// Mitsubishi GX Works2 project: 機電整合乙級第五題-ST   PLC: FX3U/FX3UC

// task Task_01 (event TRUE, interval 0, priority 31): POU_01

PROGRAM POU_01
VAR
  wProgramStep : INT;
  ldStore : R_TRIG;
  ldFetch : R_TRIG;
  wHighSpeed : INT;
  wLowSpeed : INT;
  wXPos : INT;
  tdT22 : TON;
END_VAR
VAR CONSTANT
  dwLEVEL1 : INT := 100;
END_VAR
VAR
  tdT23 : TON;
  wCellNo : INT;
  rtX10 : R_TRIG;
  tdT27 : TON;
  wZPos : INT;
  tdT29 : TON;
  ftX10 : F_TRIG;
  tdT33 : TON;
  tdT41 : TON;
  tdT42 : TON;
  tdT43 : TON;
  bOutbound : BOOL;
  tdT21 : TON;
  wXNext : INT;
  wXCurr : INT;
  bM17 : BOOL;
  bM143 : BOOL;
  tdT143 : TON;
  tdT144 : TON;
END_VAR
(* 機電整合乙級術科第五題
   Author: Steven Luo
   Date: 2018/10/25
*)

IF M8000 THEN
	WR3A(TRUE, 0, 21, D53);
	M8026 := TRUE;
END_IF;

IF M8002 THEN
	OUT_C(TRUE, CC251, K999999);
	wLowSpeed := 1200;
	wHighSpeed := 4000;
	D53 := wLowSpeed;
	wProgramStep := 0;
END_IF;

IF NOT X17 THEN (* 急停 *)
	ZRST(TRUE, Y0, Y7);
	ZRST(TRUE, D0, D50);
	ZRST(TRUE, M130, M144);
	ZRST(TRUE, M150, M153);
	D5 := 513;
	bM17 := TRUE;
	wProgramStep := 0;
END_IF;

IF X17 AND bM17 AND M132 THEN (* 解除急停，按下復歸 *)
	bM17 := FALSE;
	bM143 := TRUE;
	tdT143(IN := FALSE);
	tdT144(IN := FALSE);
	wProgramStep := 100;
END_IF;

IF bM143 THEN (* 黃燈閃爍 *)
	tdT143(IN := NOT tdT144.Q, PT := T#500ms);
	tdT144(IN := tdT143.Q, PT := T#500ms);
	M143 := tdT143.Q;
END_IF;

CASE wProgramStep OF
0:
	IF X17 THEN
		IF M130 THEN
			wProgramStep := 200;
		ELSE
			wProgramStep := 20;
		END_IF;
	END_IF;
20:
	IF M130 THEN
		wProgramStep := 0;
	END_IF;
	IF WORD_TO_INT(D0) > 0 THEN
		ldStore(_CLK := M135);
		ldFetch(_CLK := M136);
		IF ldStore.Q THEN
			IF D10 = 0 THEN
				D10 := D0;
			ELSIF (D11 = 0) AND (D0 <> D10) THEN
				D11 := D0;
			ELSIF (D12 = 0) AND (D0 <> D10) AND (D0 <> D11) THEN
				D12 := D0;
			END_IF;
			D0 := 0;
		END_IF;
		IF ldFetch.Q THEN
			IF D30 = 0 THEN
				D30 := D0;
			ELSIF (D31 = 0) AND (D0 <> D30) THEN
				D31 := D0;
			ELSIF (D32 = 0) AND (D0 <> D30) AND (D0 <> D31) THEN
				D32 := D0;
			END_IF;
			D0 := 0;
		END_IF;
	END_IF;
	IF M137 THEN
		D10 := 0;
		D11 := 0;
		D12 := 0;
		M152 := FALSE;
	END_IF;
	IF M138 THEN
		D30 := 0;
		D31 := 0;
		D32 := 0;
		M153 := FALSE;
	END_IF;
	IF M150 AND WORD_TO_INT(D10) > 0 THEN
		M152 := TRUE;
		M153 := FALSE;
	END_IF;
	IF M151 AND WORD_TO_INT(D30) > 0 THEN
		M152 := FALSE;
		M153 := TRUE;
	END_IF;
	IF X2 AND X4 AND X5 AND X6 THEN (* 原點條件 *)
		D5 := 0;
		IF M131 THEN
			wXPos := 0;
			wZPos := 0;
			wCellNo := 0;
			wXCurr := 0;
			tdT21(IN := FALSE);
			tdT22(IN := FALSE);
			tdT23(IN := FALSE);
			tdT27(IN := FALSE);
			tdT29(IN := FALSE);
			tdT33(IN := FALSE);
			tdT41(IN := FALSE);
			tdT42(IN := FALSE);
			tdT43(IN := FALSE);
			D5 := 510;
			IF M152 THEN (* 存料 *)
				wProgramStep := 21;
			ELSIF M153 THEN (* 取料 *)
				wProgramStep := 40;
			END_IF;
		END_IF;
	END_IF;
21:
	Y11 := TRUE;
	IF X3 THEN (* 進料感測 *)
		Y11 := FALSE;
		tdT21(IN := TRUE, PT := T#500ms);
		IF tdT21.Q THEN
			wProgramStep := 22;
		END_IF;
	END_IF;
22:
	Y6 := TRUE; (* Y軸伸前 *)
	IF X7 THEN (* Y軸前位 *)
		D5 := 511;
		Y7 := TRUE; (* D+氣壓夾爪夾 *)
		tdT22(IN := TRUE, PT := T#500ms);
		IF tdT22.Q THEN
			wProgramStep := 23;
		END_IF;
	END_IF;
23:
	Y3 := TRUE; (* Z軸上升 *)
	tdT23(IN := TRUE, PT := T#500ms);
	IF tdT23.Q THEN
		Y3 := FALSE;
		wProgramStep := 24;
	END_IF;
24:
	Y6 := FALSE; (* Y軸縮回 *)
	IF X6 THEN (* Y軸後位 *)
		D5 := 0;
		wProgramStep := 25;
	END_IF;
25:
	Y5 := TRUE; (* Z軸下降 *)
	IF X5 THEN
		Y5 := FALSE;
		wProgramStep := 26;
	END_IF;
26:
	IF WORD_TO_INT(D10) > 0 THEN
		wCellNo := D10;
		D10 := 0;
	ELSIF WORD_TO_INT(D11) > 0 THEN
		wCellNo := D11;
		D11 := 0;
	ELSIF WORD_TO_INT(D12) > 0 THEN
		wCellNo := D12;
		D12 := 0;
	END_IF;
	wXPos := wCellNo MOD 10;
	(* Z軸座標為C251數值 *)
	wZPos := dwLEVEL1 + (wCellNo / 10 - 1) * 1600;
	IF wXPos > 0 THEN
		D60 := 0;
		wProgramStep := 27;
	ELSE
		wProgramStep := 20;
	END_IF;
27:
	Y0 := TRUE; (* X軸右移 *)
	rtX10( _CLK := X10);
	IF rtX10.Q THEN
		wXPos := wXPos - 1;
	END_IF;
	IF wXPos = 1 THEN
		RAMP(TRUE, wHighSpeed, wLowSpeed, 50, D53);
	ELSIF wXPos = 0 THEN
		Y0 := FALSE;
		Y1 := TRUE; (* X軸停止 *)
		tdT27(IN := TRUE, PT := T#500ms);
		IF tdT27.Q THEN
			Y1 := FALSE;
			wProgramStep := 28;
		END_IF;
	ELSE
		RAMP(TRUE, wLowSpeed, wHighSpeed, 50, D60);
		D53 := D60;
	END_IF;
28:
	Y3 := TRUE; (* Z軸上升 *)
	IF CN251 >= INT_TO_DINT(wZPos) THEN
		Y3 := FALSE;
		IF M152 THEN
			wProgramStep := 29;
		ELSIF M153 THEN
			wProgramStep := 41;
		END_IF;
	END_IF;
29:
	Y6 := TRUE; (* Y軸伸前 *)
	IF X7 THEN (* Y軸前位 *)
		D5 := 511;
		Y7 := FALSE;
		Y10 := TRUE; (* D-氣壓夾爪放 *)
		tdT29(IN := TRUE, PT := T#300ms);
		IF tdT29.Q THEN
			Y10 := FALSE;
			IF M153 THEN
				bOutbound := TRUE;
			END_IF;
			wProgramStep := 30;
		END_IF;
	END_IF;
30:
	Y6 := FALSE; (* Y軸縮回 *)
	IF X6 THEN (* Y軸後位 *)
		D5 := 0;
		D60 := 0;
		IF M152 THEN
			wProgramStep := 31;
		ELSIF M153 THEN
			IF bOutbound THEN
				wProgramStep := 44;
			ELSE
				wProgramStep := 31;
			END_IF;
		END_IF;
	END_IF;
31:
	Y5 := TRUE; (* Z軸下降 *)
	IF X5 THEN
		Y5 := FALSE;
		wXPos := wCellNo MOD 10;
		IF M152 THEN
			wProgramStep := 32;
		ELSIF M153 THEN
			wXPos := (5 - wXPos) + 1;
			wProgramStep := 42;
		END_IF;
	END_IF;
32:
	Y2 := TRUE; (* X軸左移 *)
	ftX10(_CLK := X10);
	IF ftX10.Q THEN
		wXPos := wXPos - 1;
	END_IF;
	IF wXPos = 0 THEN
		RAMP(TRUE, wHighSpeed, wLowSpeed, 50, D53);
	ELSE
		RAMP(TRUE, wLowSpeed, wHighSpeed, 50, D60);
		D53 := D60;
	END_IF;
	IF X4 THEN
		Y2 := FALSE;
		Y1 := TRUE; (* X軸停止 *)
		wProgramStep := 33;
	END_IF;
33:
	tdT33(IN := TRUE, PT := T#300ms);
	IF tdT33.Q THEN
		Y1 := FALSE;
		tdT21(IN := FALSE);
		tdT22(IN := FALSE);
		tdT23(IN := FALSE);
		tdT27(IN := FALSE);
		tdT29(IN := FALSE);
		tdT33(IN := FALSE);
		tdT41(IN := FALSE);
		tdT42(IN := FALSE);
		tdT43(IN := FALSE);
		IF M152 THEN
			IF (D10 = 0) AND (D11 = 0) AND (D12 = 0) THEN
				wProgramStep := 34;
			ELSE
				wProgramStep := 21; (* 繼續進料 *)
			END_IF;
		ELSIF M153 THEN
			IF (D30 = 0) AND (D31 = 0) AND (D32 = 0) THEN
				M153 := FALSE;
				wProgramStep := 20;
			ELSE
				wProgramStep := 40; (* 繼續出料 *)
			END_IF;
		END_IF;
	END_IF;
34:
	Y12 := TRUE; (* 進料座下降 *)
	IF X2 THEN (* 進料原點極限 *)
		Y12 := FALSE;
		M152 := FALSE;
		wProgramStep := 20;
	END_IF;
40:
	IF WORD_TO_INT(D30) > 0 THEN
		wCellNo := D30;
		IF WORD_TO_INT(D31) > 0 THEN
			wXNext := D31;
		ELSE
			wXNext := 0;
		END_IF;
		D30 := 0;
	ELSIF WORD_TO_INT(D31) > 0 THEN
		wCellNo := D31;
		IF WORD_TO_INT(D32) > 0 THEN
			wXNext := D32;
		ELSE
			wXNext := 0;
		END_IF;
		D31 := 0;
	ELSIF WORD_TO_INT(D32) > 0 THEN
		wCellNo := D32;
		wXNext := 0;
		D32 := 0;
	END_IF;
	wXPos := wCellNo MOD 10 - wXCurr;
	(* Z軸座標為C251數值 *)
	wZPos := dwLEVEL1 + (wCellNo / 10 - 1) * 1600 - 100;
	IF wCellNo > 0 THEN
		D60 := 0;
		bOutbound := FALSE;
		wProgramStep := 27;
	ELSE
		wProgramStep := 20;
	END_IF;
41:
	Y6 := TRUE; (* Y軸伸前 *)
	IF X7 THEN (* Y軸前位 *)
		D5 := 511;
		Y7 := TRUE; (* D+氣壓夾爪夾 *)
		tdT41(IN := TRUE, PT := T#300ms);
		IF tdT41.Q THEN
			wProgramStep := 30;
		END_IF;
	END_IF;
42:
	Y3 := TRUE; (* Z軸上升 *)
	tdT42(IN := TRUE, PT := T#1s);
	IF tdT42.Q THEN
		Y3 := FALSE;
		wProgramStep := 43;
	END_IF;
43:
	Y0 := TRUE; (* X軸右移 *)
	ftX10( _CLK := X10);
	IF ftX10.Q THEN
		wXPos := wXPos - 1;
	END_IF;
	IF wXPos = 1 THEN
		RAMP(TRUE, wHighSpeed, wLowSpeed, 50, D53);
	ELSIF wXPos = 0 THEN
		Y0 := FALSE;
		Y1 := TRUE; (* X軸停止 *)
		tdT43(IN := TRUE, PT := T#500ms);
		IF tdT43.Q THEN
			Y1 := FALSE;
			wProgramStep := 29;
		END_IF;
	ELSE
		RAMP(TRUE, wLowSpeed, wHighSpeed, 50, D60);
		D53 := D60;
	END_IF;
44:
	Y5 := TRUE; (* Z軸下降 *)
	IF X5 THEN
		Y5 := FALSE;
		wXCurr := wXNext MOD 10;
		wXPos := 6 - wXCurr;
		IF wXNext = 0 THEN
			wProgramStep := 32;
		ELSE
			wProgramStep := 45;
		END_IF;
	END_IF;
45:
	Y2 := TRUE; (* X軸左移 *)
	rtX10( _CLK := X10);
	IF rtX10.Q THEN
		wXPos := wXPos - 1;
	END_IF;
	IF wXPos = 1 THEN
		RAMP(TRUE, wHighSpeed, wLowSpeed, 50, D53);
	ELSIF wXPos = 0 THEN
		Y2 := FALSE;
		Y1 := TRUE; (* X軸停止 *)
		tdT43(IN := TRUE, PT := T#500ms);
		IF tdT43.Q THEN
			Y1 := FALSE;
			wProgramStep := 33;
		END_IF;
	ELSE
		RAMP(TRUE, wLowSpeed, wHighSpeed, 50, D60);
		D53 := D60;
	END_IF;
100:
	D5 := 512;
	D53 := wLowSpeed;
	Y6 := FALSE;
	IF X6 THEN
		Y5 := TRUE;
		IF X5 THEN
			Y5 := FALSE;
			Y2 := TRUE;
			IF X4 THEN
				Y2 := FALSE;
				Y12 := TRUE;
				IF X2 THEN
					Y12 := FALSE;
					D5 := 0;
					bM143 := FALSE;
					M143 := FALSE;
					wProgramStep := 0;
				END_IF;
			END_IF;
		END_IF;
	END_IF;
200:
	IF X6 THEN
		D5 := 0;
		OUT(M110, Y2); (* X軸左移 *)
		OUT(M111, Y0); (* X軸右移 *)
		OUT(M112, Y3); (* Z軸上升 *)
		OUT(M113, Y5); (* Z軸下降 *)
		IF X5 THEN
			CN251 := 0;
		END_IF;
	END_IF;
	IF M114 THEN (* 水平缸伸出 *)
		Y6 := TRUE;
	END_IF;
	IF M115 THEN (* 水平缸縮回 *)
		Y6 := FALSE;
	END_IF;
	OUT(M116, Y7); (* 夾爪夾 *)
	OUT(M117, Y10); (* 夾爪放 *)
	OUT(M118, Y11); (* 進料座上升 *)
	OUT(M119, Y12); (* 進料座下降 *)
	IF NOT M130 THEN
		wProgramStep := 0;
	END_IF;
END_CASE;
END_PROGRAM
